PROGRAM StatesExample
VAR
END_VAR

PackMLExample();

END_PROGRAM

(* stored: Version 1.1.0.1
   POU StatesExample: Id {78e76905-38c3-4db6-8fcd-815a0d681fdb}, SpecialFunc None *)
